Staubli VAL3: VALCLEAN.dtx


